FUNCTION_BLOCK PICKUP_SCREW_SEQ
VAR_IN_OUT
	xExecute:		BOOL;
END_VAR
VAR_OUTPUT
	xDone:			BOOL;
END_VAR
VAR
	tpReset:			TP;
	rtDone:				R_TRIG;
	rtExecute:			R_TRIG;
	ftTimePulse:		F_TRIG;
	tpTimePulse:		TP;
	lrTargetPos:		LREAL;
	xTransCondition:	BOOL;	
	xTransRelease:		BOOL;
	SFCInit:			BOOL;
	SFCReset:			BOOL;	
	SFCError:			BOOL;
END_VAR

rtDone(CLK:=xDone);
IF rtDone.Q THEN
	xTransRelease:=FALSE;	
	SFCReset:=TRUE;
END_IF

rtExecute(CLK:=xExecute);
IF rtExecute.Q THEN
	xTransRelease:=TRUE;
	SFCReset:=FALSE;
END_IF

IF xExecute THEN
	aSEQ_ACT();
END_IF

tpReset(IN:=SFCError, PT:=T#250MS);
SFCReset:= tpReset.Q;

ACTION ACK_DONE_AXIS_active:
IF G_sAxisDone.X OR G_sAxisDone.Y OR G_sAxisDone.Z OR G_sAxisDone.c THEN
	G_sAckAxisDone.X:=TRUE;
	G_sAckAxisDone.Y:=TRUE;
	G_sAckAxisDone.Z:=TRUE;
	G_sAckAxisDone.C:=TRUE;
ELSE
	G_sAckAxisDone.X:=FALSE;
	G_sAckAxisDone.Y:=FALSE;
	G_sAckAxisDone.Z:=FALSE;
	G_sAckAxisDone.C:=FALSE;
END_IF

xTransCondition:= NOT G_sAckAxisDone.X AND NOT G_sAckAxisDone.Y AND NOT G_sAckAxisDone.Z AND NOT G_sAckAxisDone.C;
END_ACTION

ACTION aSEQ_ACT:
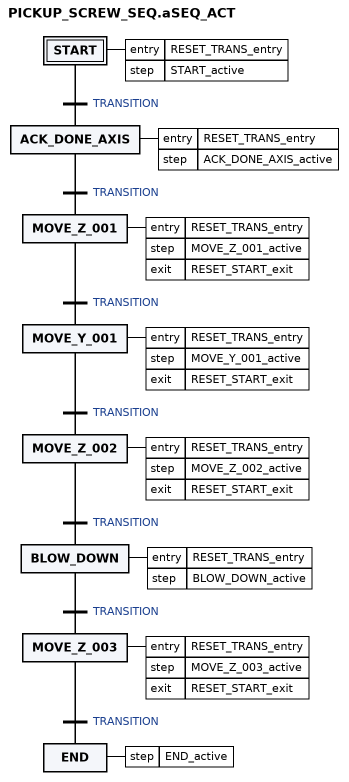
INITIAL_STEP START:
    RESET_TRANS_entry(P1);  // entry action
    START_active(N);  // step action
END_STEP
TRANSITION FROM START TO ACK_DONE_AXIS
    := TRANSITION;
END_TRANSITION
STEP ACK_DONE_AXIS:
    RESET_TRANS_entry(P1);  // entry action
    ACK_DONE_AXIS_active(N);  // step action
END_STEP
TRANSITION FROM ACK_DONE_AXIS TO MOVE_Z_001
    := TRANSITION;
END_TRANSITION
STEP MOVE_Z_001:
    RESET_TRANS_entry(P1);  // entry action
    MOVE_Z_001_active(N);  // step action
    RESET_START_exit(P0);  // exit action
END_STEP
TRANSITION FROM MOVE_Z_001 TO MOVE_Y_001
    := TRANSITION;
END_TRANSITION
STEP MOVE_Y_001:
    RESET_TRANS_entry(P1);  // entry action
    MOVE_Y_001_active(N);  // step action
    RESET_START_exit(P0);  // exit action
END_STEP
TRANSITION FROM MOVE_Y_001 TO MOVE_Z_002
    := TRANSITION;
END_TRANSITION
STEP MOVE_Z_002:
    RESET_TRANS_entry(P1);  // entry action
    MOVE_Z_002_active(N);  // step action
    RESET_START_exit(P0);  // exit action
END_STEP
TRANSITION FROM MOVE_Z_002 TO BLOW_DOWN
    := TRANSITION;
END_TRANSITION
STEP BLOW_DOWN:
    RESET_TRANS_entry(P1);  // entry action
    BLOW_DOWN_active(N);  // step action
END_STEP
TRANSITION FROM BLOW_DOWN TO MOVE_Z_003
    := TRANSITION;
END_TRANSITION
STEP MOVE_Z_003:
    RESET_TRANS_entry(P1);  // entry action
    MOVE_Z_003_active(N);  // step action
    RESET_START_exit(P0);  // exit action
END_STEP
TRANSITION FROM MOVE_Z_003 TO END
    := TRANSITION;
END_TRANSITION
STEP END:
    END_active(N);  // step action
END_STEP
END_ACTION

ACTION BLOW_DOWN_active:
tpTimePulse(IN:=NOT tpTimePulse.Q, PT:=T#3000MS);
ftTimePulse(CLK:=tpTimePulse.Q);
xTransCondition:= ftTimePulse.Q;
END_ACTION

ACTION END_active:
xDone:=TRUE;
xTransCondition:=FALSE;
END_ACTION

ACTION MOVE_Y_001_active:
G_sTargetPosition.Y:= G_asIndividualAxisPositions[CE_AXIS_Y].Positions[1].Target;
G_sStartToPos.Y:= TRUE;

xTransCondition:= G_sAxisDone.Y;
END_ACTION

ACTION MOVE_Z_001_active:
G_sTargetPosition.Z:= G_asIndividualAxisPositions[CE_AXIS_Z].Positions[1].Target;
G_sStartToPos.Z:= TRUE;

xTransCondition:= G_sAxisDone.Z;
END_ACTION

ACTION MOVE_Z_002_active:
G_sTargetPosition.Z:= G_asIndividualAxisPositions[CE_AXIS_Z].Positions[2].Target;
G_sStartToPos.Z:= TRUE;

xTransCondition:= G_sAxisDone.Z;
END_ACTION

ACTION MOVE_Z_003_active:
G_sTargetPosition.Z:= G_asIndividualAxisPositions[CE_AXIS_Z].Positions[1].Target;
G_sStartToPos.Z:= TRUE;

xTransCondition:= G_sAxisDone.Z;
END_ACTION

ACTION RESET_START_exit:
IF G_sAxisDone.X OR G_sAxisDone.Y OR G_sAxisDone.Z OR G_sAxisDone.c THEN
	G_sAckAxisDone.X:=TRUE;
	G_sAckAxisDone.Y:=TRUE;
	G_sAckAxisDone.Z:=TRUE;
	G_sAckAxisDone.C:=TRUE;
ELSE
	G_sAckAxisDone.X:=FALSE;
	G_sAckAxisDone.Y:=FALSE;
	G_sAckAxisDone.Z:=FALSE;
	G_sAckAxisDone.C:=FALSE;
	
	G_sStartToPos.X:=FALSE;
	G_sStartToPos.Y:=FALSE;
	G_sStartToPos.Z:=FALSE;
	G_sStartToPos.C:=FALSE;
END_IF
END_ACTION

ACTION RESET_TRANS_entry:
xTransCondition:= false;
END_ACTION

ACTION START_active:
xDone:=FALSE;
xTransCondition:= NOT xDone;
END_ACTION

TRANSITION TRANSITION:
xTransRelease AND xTransCondition
END_TRANSITION

END_FUNCTION_BLOCK

(* stored: Version 1.1.0.1, ProductVersion 3.1.4022.18
   POU PICKUP_SCREW_SEQ: Id {94535a87-f883-4a98-950a-4781d79e809f}, SpecialFunc None
   Folder xActive: Id {e4027299-5cd7-43ec-b143-156e866d2f63}
   Folder xEntry: Id {385eee8e-6deb-493d-ac0d-7d712c389015}
   Folder xExit: Id {10a7a315-5933-45f9-8c7b-8232d0988c3c}
   Folder xTrans: Id {1a17d362-dec9-4878-995d-f0a87485e6d1}
   Action ACK_DONE_AXIS_active: Id {2ecc881f-1f41-45ea-99e3-e5c9752bc232}
   Action aSEQ_ACT: Id {d454e913-e664-4eb9-a0a9-87dfb70f96de}
   Action BLOW_DOWN_active: Id {0124ca8f-048d-45f3-9b0f-929e09226d7b}
   Action END_active: Id {1b630793-fdcc-43aa-b546-9cfb2c5ba0f6}
   Action MOVE_Y_001_active: Id {7df994c1-8f33-46d7-8f08-8a7c418089b2}
   Action MOVE_Z_001_active: Id {0b414e00-a49f-4a20-8315-69fc64f98d59}
   Action MOVE_Z_002_active: Id {fbc3cd7a-de93-48ce-8770-c413b8e6f4a3}
   Action MOVE_Z_003_active: Id {07d27959-981f-42d3-97c5-2201ff3bce0b}
   Action RESET_START_exit: Id {9139992c-614b-4d69-bf99-580bd29393a5}
   Action RESET_TRANS_entry: Id {09d325b3-df2b-471d-bced-a71d78a761c8}
   Action START_active: Id {f87d9745-6d5a-4813-a510-9edc114ba0b3}
   Transition TRANSITION: Id {b8563804-5471-46ce-b574-9edf0aa9aa82} *)
